FUNCTION_BLOCK STATION2_INFO
  {SET_ATTRIBUTE(OpcUa, SERVICE)}
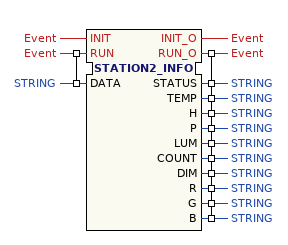
  EVENT_INPUT
    INIT;
    RUN WITH DATA; {SET_ATTRIBUTE(OpcUa, Method)}
  END_EVENT
  EVENT_OUTPUT
    INIT_O;
    RUN_O WITH STATUS, TEMP, H, P, LUM, COUNT, DIM, R, G, B;
  END_EVENT
  VAR_INPUT
    DATA : STRING;
  END_VAR
  VAR_OUTPUT
    STATUS : STRING;
    TEMP : STRING;
    H : STRING;
    P : STRING;
    LUM : STRING;
    COUNT : STRING;
    DIM : STRING;
    R : STRING;
    G : STRING;
    B : STRING;
  END_VAR
END_FUNCTION_BLOCK
